{attribute 'OPC.UA.DA.JobMethod' := 'MyJob'}
FUNCTION_BLOCK FB_Job
VAR
	// Used for debugging purposes to display InputArguments of method call
	Input_a : INT; // used to store InputArg "a" from Start() method
	Input_b : LREAL; // used to store InputArg "b" from Start() method
	Input_c : BOOL; // used to store InputArg "c" from Start() method
	Input_d : ST_Complex_1; // used to store InputArg "d" from Start() method
	callCounterStart : ULINT; // counts how many times the Start() method has been called
	callCounterCheckState : ULINT; // counts how many times the CheckState() method has been called
	callCounterAbort : ULINT; // counts how many times the Abort() method has been called
	
	// Timer to "artificially delay" job execution
	timer : TON := (PT:=T#4S);
	
	// Variables to determine if a job has been started (Start() method has been called) or finished
	jobRunning : BOOL;
	jobFinished : BOOL;

	// State machine variable
	state : UDINT;
END_VAR

CASE state OF
	0:
		IF jobRunning THEN
			state := state + 1;
		END_IF
		
	1:
		timer(IN:=TRUE);
		IF timer.Q THEN
			timer(IN:=FALSE);
			jobRunning := FALSE;
			jobFinished := TRUE;
			state := 0;
		END_IF
		
END_CASE

{attribute 'TcRpcEnable' := '1'}
METHOD Abort : HRESULT
VAR_INPUT
	hdl : UDINT; // Do not change, used by server.
END_VAR
callCounterAbort := callCounterAbort + 1;
END_METHOD

{attribute 'TcRpcEnable' := '1'}
METHOD CheckState : HRESULT
VAR_INPUT
	hdl : UDINT; // Do not change, used by server.
END_VAR
VAR_OUTPUT
	bBusy : BOOL; // Do not change. Used by server to find out if the job is finished
	
	// List of OutputArguments for OPC UA method, may be customized
	a : INT; // some description
	b : LREAL; // some description
	c : BOOL; // some description
	d : ST_Complex_1; // some description
END_VAR
callCounterCheckState := callCounterCheckState + 1;
IF NOT jobFinished THEN
	bBusy := TRUE; // job is not finished yet
	CheckState := 0; // no error
ELSE
	bBusy := FALSE; // job is finished
	CheckState := 0; // done, no error occured during execution (OPC UA StatusCode "GOOD")
	jobFinished := FALSE;
	a := Input_a;
	b := Input_b;
	c := Input_c;
	d := Input_d;
END_IF
END_METHOD

{attribute 'TcRpcEnable' := '1'}
METHOD Start : HRESULT
VAR_INPUT
	// List of InputArguments for OPC UA method, may be customized
	a : INT; // some description
	b : LREAL; // some description
	c : BOOL; // some description
	d : ST_Complex_1; // some description
END_VAR
VAR_OUTPUT
	hdl : UDINT; // Do not change, used by server.
END_VAR
callCounterStart := callCounterStart + 1;
Input_a := a;
Input_b := b;
Input_c := c;
Input_d := d;
jobRunning := TRUE;
Start := 0; // no error occured, e.g. while parsing the input arguments (0 = OPC UA StatusCode "GOOD")
END_METHOD

END_FUNCTION_BLOCK

(* stored: Version 1.1.0.1, ProductVersion 3.1.4024.11
   POU FB_Job: Id {8a26e45c-b764-4450-92ac-a1261a1e29af}, SpecialFunc None
   Method Abort: Id {a3f18e5a-12e6-4a70-8697-275827ac76ca}
   Method CheckState: Id {89e7ee9d-9129-44d6-b390-8e15e88d0e04}
   Method Start: Id {d7456b05-1ddc-4259-b442-8ae76bbb795d} *)
